{attribute addProperty BoxType "EL5151-0000-0016"}
{attribute addProperty Id "ENC_InputsAT %I*ENC_Inputs_2D5D285780100ENC_Inputs_1AT %I*ENC_Inputs_AC51B8A03240ENC_OutputsAT %Q*ENC_Outputs_90374C536480WcStateAT %I*WcState_F855686C1620InfoDataAT %I*InfoData_BC63D37F80100"}
{attribute addProperty CRC "2243964890"}
{attribute addProperty SizeInBites "272"}
{attribute addProperty SizeInBytes "34"}
TYPE EL5151_04803048 :
STRUCT
	{attribute addProperty Name "ENC_Inputs"}
	ENC_Inputs : ENC_Inputs_2D5D2857;
	{attribute addProperty Name "ENC_Inputs_1"}
	ENC_Inputs_1 : ENC_Inputs_AC51B8A0;
	{attribute addProperty Name "ENC_Outputs"}
	ENC_Outputs : ENC_Outputs_90374C53;
	{attribute addProperty Name "WcState"}
	WcState : WcState_F855686C;
	{attribute addProperty Name "InfoData"}
	InfoData : InfoData_BC63D37F;
END_STRUCT
END_TYPE

(* stored: Version 1.2.0.0, ProductVersion 3.1.4024.9
   DUT EL5151_04803048: Id {31d305fd-d69c-4db4-ad42-94815f79a2e6} *)
